RoboDK station: fairino_dk_test.rdk

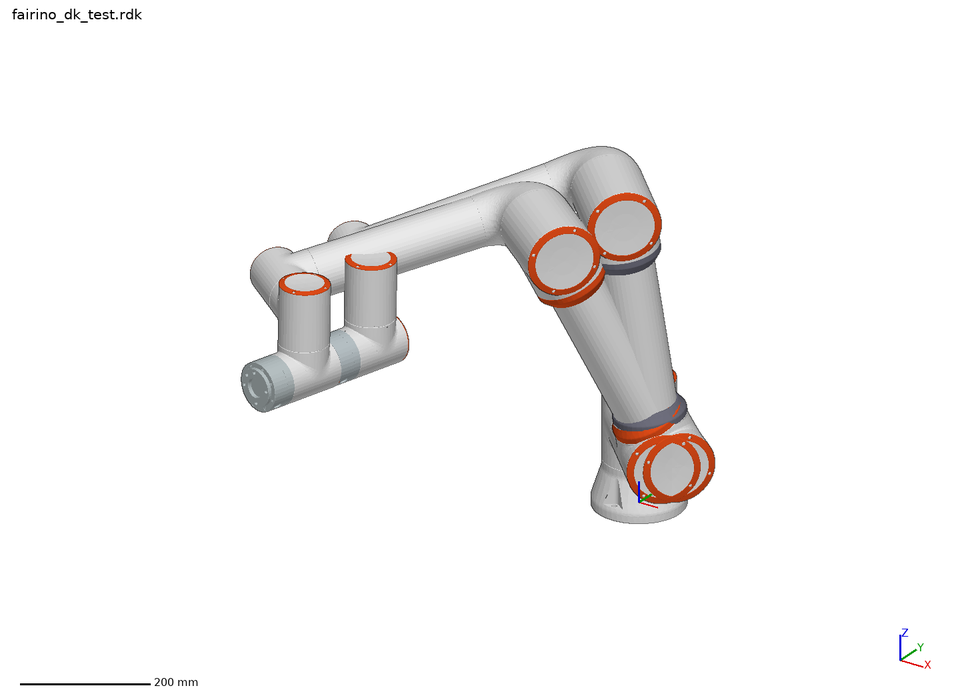
[picture v0: the station drawn from its stored meshes, robots at their saved joint values, targets as dots, program paths as lines]
Station fairino_dk_test (saved by RoboDK 5.9.2). Poses are relative to the parent item; angles as X-Y-Z fixed-axis rotations.
  - frame FAIRINO FR5 Base at (0, 0, 0) mm
    - robot FAIRINO FR3 WML offset (model FAIRINO FR5): 6 axes
        modified DH rows (alpha deg, a mm, theta deg, d mm): 0, 0, 0, 152; 90, 0, 180, 0; 0, 425, 0, 0; 0, 395, 0, 102; -90, 0, 0, 102; 90, 0, 180, 100
        joint limits [-175, -265, -160, -265, -175, -355] to [175, 85, 160, 85, 175, 355]; home [0, -90, -90, 0, 90, 0]; saved at [45.977, -81.678, 98.089, -17.306, 59.288, 51.038]
    - robot FAIRINO FR3 WML (model FAIRINO FR5): 6 axes
        modified DH rows (alpha deg, a mm, theta deg, d mm): 0, 0, 0, 152; 90, 0, 180, 0; 0, 425, 0, 0; 0, 395, 0, 102; -90, 0, 0, 102; 90, 0, 180, 100
        joint limits [-175, -265, -160, -265, -175, -355] to [175, 85, 160, 85, 175, 355]; home [0, -90, -90, 0, 90, 0]; saved at [52.94, -64.045, 74.586, -11.382, 66.25, 50.92]
  - Python program Prog2 (listed below)

--- Python program Prog2 ---
from robodk import robolink    # RoboDK API
from robodk import robomath    # Robot toolbox
from pythonosc import udp_client
from pythonosc.osc_server import BlockingOSCUDPServer
from pythonosc.dispatcher import Dispatcher

# --- Configuration ---
ROBOT_NAME = 'FAIRINO FR3 WML'
ROBOT_OFFSET_NAME = 'FAIRINO FR3 WML offset' # Added second robot name
OSC_IN_IP = "127.0.0.1"
OSC_IN_PORT = 8100
OSC_OUT_IP = "127.0.0.1"
OSC_OUT_PORT = 9100

# Latest TCP adjustment [x, y, z, rx, ry, rz]
tcp_offset_vals = [0.0] * 6

# Initialize RoboDK
RDK = robolink.Robolink()
robot = RDK.Item(ROBOT_NAME, robolink.ITEM_TYPE_ROBOT)
robot_preview = RDK.Item(ROBOT_OFFSET_NAME, robolink.ITEM_TYPE_ROBOT) # Added second robot item
client = udp_client.SimpleUDPClient(OSC_OUT_IP, OSC_OUT_PORT)

def handle_offset(address, *args):
    global tcp_offset_vals
    tcp_offset_vals = [float(a) for a in args[:6]]

def handle_joints(address, *args):
    # 1. Capture incoming joints
    in_joints = [float(a) for a in args]

    # 2. Update virtual robot viewport
    robot.setJoints(in_joints)

    # 3. Forward Kinematics
    current_pose = robot.SolveFK(in_joints)

    # 4. Create offset matrix (Standard XYZ ABC)
    offset_matrix = robomath.KUKA_2_Pose(tcp_offset_vals)

    # 5. Apply offset relative to BASE (Offset * Pose)
    # Swapping the order here changes it from Tool Space to Base Space
    target_pose =  offset_matrix * current_pose

    # 6. Solve for new joints
    new_joints = robot.SolveIK(target_pose, in_joints)

    # Check if the result is valid
    if new_joints.size(0) > 0:
        raw_list = new_joints.tolist()

        if isinstance(raw_list[0], list):
            out_joints = [j[0] for j in raw_list]
        else:
            out_joints = raw_list

        robot_preview.setJoints(out_joints)
        client.send_message("/robot/adjusted_joints", out_joints)
    else:
        print("IK Solve Failed: Position likely out of reach.")


# --- OSC Server Setup ---
dispatcher = Dispatcher()
dispatcher.map("/joints", handle_joints)
dispatcher.map("/offset", handle_offset)

print(f"Kinematics Engine Running...")
print(f"Listening: {OSC_IN_IP}:{OSC_IN_PORT} -> Sending: {OSC_OUT_PORT}")
server = BlockingOSCUDPServer((OSC_IN_IP, OSC_IN_PORT), dispatcher)
server.serve_forever()
